# EPICS StreamDevice protocol: protocol/Berthold-LB6420.proto
# Berthold-LB6420.proto

# Communication protocol for Berthold LB 6420 radiation probes

# Protocol terminator character

Terminator = LF;

# Averaging time (readback)

getAveragingTime {
    out "AVERAGING_TIME?";
    in "%u";
}

# Gamma

getGamma {
    out "GAMMA?";
    in "%f";
}

# High energy neutrons

getHighEnergyNeutrons {
    out "HIGH_ENERGY_NEUTRONS?";
    in "%f";
}

# Total dose rate

getTotalDoseRate {
    out "TOTAL_DOSE_RATE?";
    in "%f";
}

# Total neutron rate

getTotalNeutronRate {
    out "TOTAL_NEUTRON_RATE?";
    in "%f";
}

# Averaging time (setpoint)

setAveragingTime {
    out "AVERAGING_TIME %u";
    in "OK";
    @init {
        getAveragingTime;
    }
}
